{attribute addProperty BoxType "EK1122-0000-0018"}
{attribute addProperty Id "Beckhoff_EKxxxx_0080sub_EK1100EK1100_179A0949162"}
{attribute addProperty CRC "1237391052"}
{attribute addProperty SizeInBites "16"}
{attribute addProperty SizeInBytes "2"}
TYPE Beckhoff_EKxxxx_0080EK1122_49C116CC EXTENDS EK1122_179A0949 :
STRUCT
	{attribute addProperty Name "Beckhoff_EKxxxx_0080sub_EK1100"}
	Beckhoff_EKxxxx_0080sub_EK1100 : EK1100_179A0949;
END_STRUCT
END_TYPE

(* stored: Version 1.2.0.0, ProductVersion 3.1.4024.9
   DUT Beckhoff_EKxxxx_0080EK1122_49C116CC: Id {dc777949-3d1e-4528-bd3b-690fd31ded59} *)
